# EPICS autosave request: ADApp/Db/andorCCD_settings.req
$(P)$(R)AndorImageMode
$(P)$(R)AndorACTInKinetics
$(P)$(R)AndorANumInKinetics
$(P)$(R)AndorFKHeight
$(P)$(R)AndorFKHBinning
$(P)$(R)AndorFKVBinning
$(P)$(R)AndorFKOffset
$(P)$(R)AndorShutterMode
$(P)$(R)AndorShutterExTTL
$(P)$(R)PALFilePath
$(P)$(R)AndorADCSpeed
